TYPE ST_FrmWcDiag :
STRUCT
	iNum					:DINT;
	sBin					:String;
END_STRUCT
END_TYPE

(* stored: Version 1.1.0.1, ProductVersion 3.1.4022.12
   DUT ST_FrmWcDiag: Id {f595fcfa-bc50-4b9c-b0f8-0243484c5712} *)
